FUNCTION Convert_UDINT_TO_TOD : Hresult
VAR_INPUT
	in : UDINT;
	out : REFERENCE TO TOD;
END_VAR
VAR
	converted : TOD;
END_VAR

converted := UDINT_TO_TOD(in);

IF (TOD_TO_UDINT(converted) <> in) THEN
	Convert_UDINT_TO_TOD := INCOMPATIBLE;
	RETURN;
END_IF

out := converted;

END_FUNCTION

(* stored: Version 1.1.0.1, ProductVersion 3.1.4024.12
   POU Convert_UDINT_TO_TOD: Id {14006796-60d2-473b-9107-c1ee0ce3215f}, SpecialFunc None *)
